SUBAPPLICATION AD_SPLIT_2_UNGATED (* Wie AD_SPLIT_2, aber OHNE Aenderungserkennung - reicht JEDES eingehende Event bedingungslos an beide Ausgaenge weiter, mit dem jeweils aktuellen Wert (auch wenn unveraendert seit dem letzten Aufruf). *)
  (* Standard: 61499-2; Description: Copyright (c) 2026 Meisterschulen am Ostbahnhof This program and the accompanying materials are made available under the terms of the Eclipse Public License 2.0 which is available at https://www.eclipse.org/legal/epl-2.0/ SPDX-License-Identifier: EPL-2.0 *)
  (* Version 1.1, 2026-08-31, Franz Höpfinger, Meisterschulen am Ostbahnhof, Noetig geworden, nachdem AD_SPLIT_2/_3 (GEN_AD_SPLIT) auf Aenderungserkennung umgestellt wurden - Verbraucher, die eine periodische Kadenz unabhaengig von Wertaenderung brauchen (z.B. FT_DERIV_AR fuer eine Frequenzberechnung), frieren sonst ein, sobald der Wert stabil bleibt. Intern: einmal entpackt (AD_D_TO_DWORD), zweimal getrennt wieder verpackt (AD_DWORD_TO_D) - direkte Boundary-zu-Boundary-Adapterverdrahtung war nicht zulaessig. *)
  PACKAGE MyLib::sys;
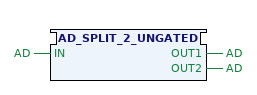
  SOCKETS
    IN : adapter::types::unidirectional::AD; (* Eingang *)
  END_SOCKETS
  PLUGS
    OUT1 : adapter::types::unidirectional::AD; (* Bedingungslose Kopie von IN *)
    OUT2 : adapter::types::unidirectional::AD; (* Bedingungslose Kopie von IN *)
  END_PLUGS
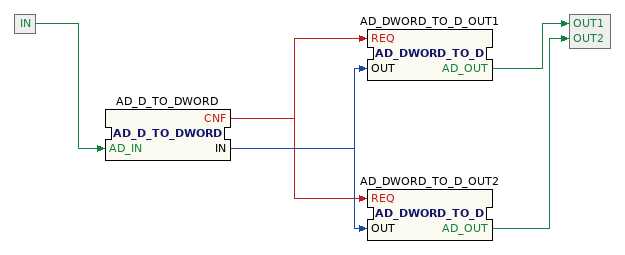
  FBS
    AD_D_TO_DWORD : adapter::conversion::unidirectional::AD_D_TO_DWORD;
    AD_DWORD_TO_D_OUT1 : adapter::conversion::unidirectional::AD_DWORD_TO_D;
    AD_DWORD_TO_D_OUT2 : adapter::conversion::unidirectional::AD_DWORD_TO_D;
  END_FBS
  EVENT_CONNECTIONS
    AD_D_TO_DWORD.CNF TO AD_DWORD_TO_D_OUT1.REQ;
    AD_D_TO_DWORD.CNF TO AD_DWORD_TO_D_OUT2.REQ;
  END_CONNECTIONS
  DATA_CONNECTIONS
    AD_D_TO_DWORD.IN TO AD_DWORD_TO_D_OUT1.OUT;
    AD_D_TO_DWORD.IN TO AD_DWORD_TO_D_OUT2.OUT;
  END_CONNECTIONS
  ADAPTER_CONNECTIONS
    IN TO AD_D_TO_DWORD.AD_IN;
    AD_DWORD_TO_D_OUT1.AD_OUT TO OUT1;
    AD_DWORD_TO_D_OUT2.AD_OUT TO OUT2;
  END_CONNECTIONS
END_SUBAPPLICATION
